// SIMATIC S7-200 project (STEP 7-Micro/WIN), CPU 221 REL 01.10

SYMBOL_TABLE USER1
start            I0.0
LS_1             I0.1
LS_2             I0.2
D1               I0.3
D2               I0.4
D3               I0.5
Pump_1           Q0.0
Pump_2           Q0.1
Heater           Q0.2
Mini_Pump        Q0.3
Conv             Q0.4
Red              Q0.5
Green            Q0.6
END_SYMBOL_TABLE

ORGANIZATION_BLOCK MAIN:OB1
TITLE=PROGRAM COMMENTS
BEGIN
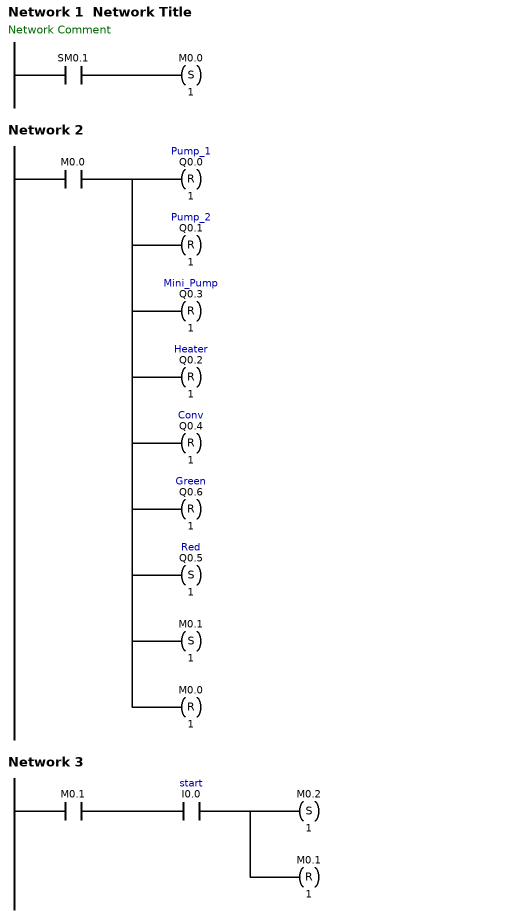
Network 1 // Network Title
// Network Comment
LD     SM0.1
S      M0.0, 1
Network 2
LD     M0.0
R      Pump_1:Q0.0, 1
R      Pump_2:Q0.1, 1
R      Mini_Pump:Q0.3, 1
R      Heater:Q0.2, 1
R      Conv:Q0.4, 1
R      Green:Q0.6, 1
S      Red:Q0.5, 1
S      M0.1, 1
R      M0.0, 1
Network 3
LD     M0.1
A      start:I0.0
S      M0.2, 1
R      M0.1, 1
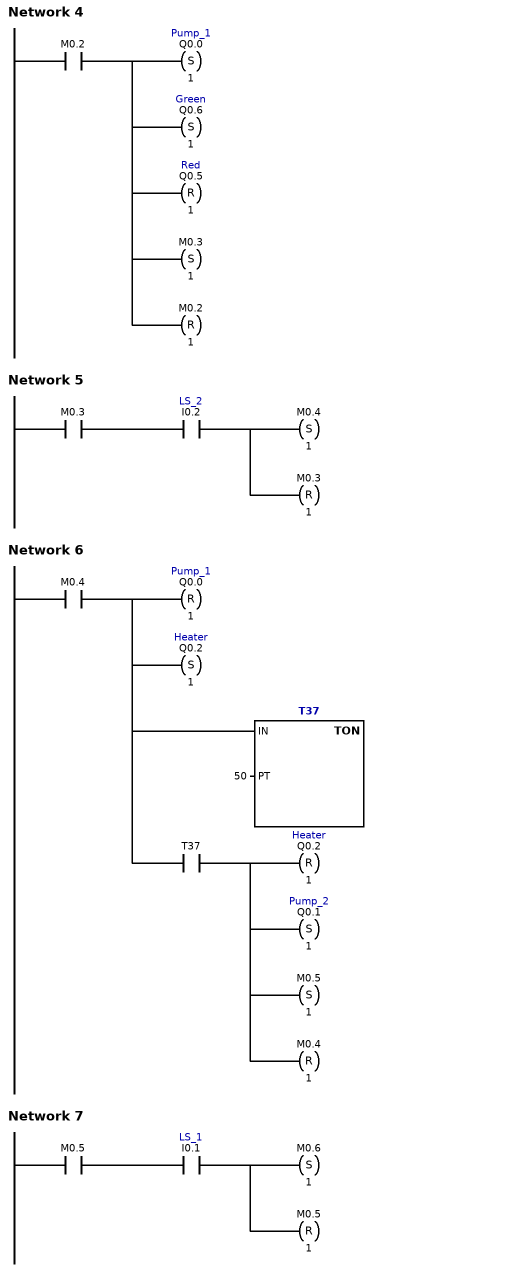
Network 4
LD     M0.2
S      Pump_1:Q0.0, 1
S      Green:Q0.6, 1
R      Red:Q0.5, 1
S      M0.3, 1
R      M0.2, 1
Network 5
LD     M0.3
A      LS_2:I0.2
S      M0.4, 1
R      M0.3, 1
Network 6
LD     M0.4
R      Pump_1:Q0.0, 1
S      Heater:Q0.2, 1
TON    T37, 50
A      T37
R      Heater:Q0.2, 1
S      Pump_2:Q0.1, 1
S      M0.5, 1
R      M0.4, 1
Network 7
LD     M0.5
A      LS_1:I0.1
S      M0.6, 1
R      M0.5, 1
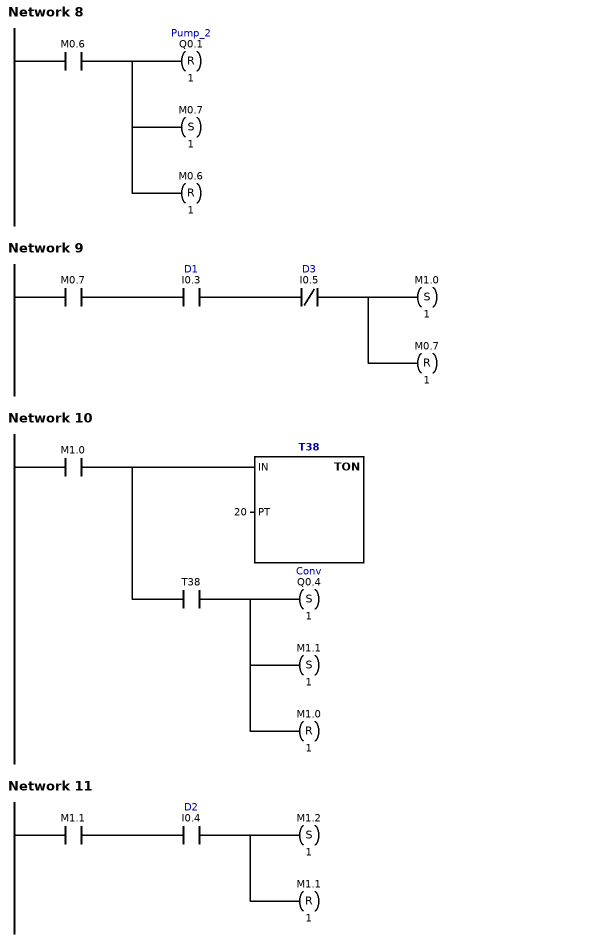
Network 8
LD     M0.6
R      Pump_2:Q0.1, 1
S      M0.7, 1
R      M0.6, 1
Network 9
LD     M0.7
A      D1:I0.3
AN     D3:I0.5
S      M1.0, 1
R      M0.7, 1
Network 10
LD     M1.0
TON    T38, 20
A      T38
S      Conv:Q0.4, 1
S      M1.1, 1
R      M1.0, 1
Network 11
LD     M1.1
A      D2:I0.4
S      M1.2, 1
R      M1.1, 1
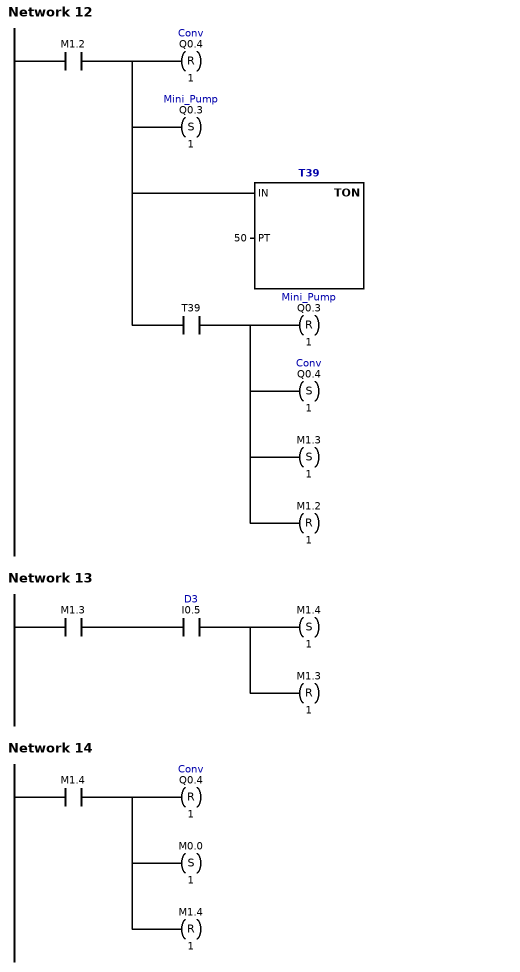
Network 12
LD     M1.2
R      Conv:Q0.4, 1
S      Mini_Pump:Q0.3, 1
TON    T39, 50
A      T39
R      Mini_Pump:Q0.3, 1
S      Conv:Q0.4, 1
S      M1.3, 1
R      M1.2, 1
Network 13
LD     M1.3
A      D3:I0.5
S      M1.4, 1
R      M1.3, 1
Network 14
LD     M1.4
R      Conv:Q0.4, 1
S      M0.0, 1
R      M1.4, 1
END_ORGANIZATION_BLOCK
